TYPE ST_CartUIData :
STRUCT
	m_joystickDataFromUI:ARRAY [0..21] OF USINT;
	m_ctrlEnableFromUI:ST_UI_control;
	m_standColumnHightLimit :LREAL;
	m_surgicalSite : UINT;
	m_surgicalLocation : UINT;
	m_cartDrapingState : UINT;
	m_cartDockingState : UINT;
	m_cartSpecificPosDocking : Vec8d;
	m_cartSpecificPosDraping : Vec8d;
END_STRUCT
END_TYPE

(* stored: Version 1.1.0.1, ProductVersion 3.1.4024.11
   DUT ST_CartUIData: Id {8a7b800d-dda3-4ddf-b29a-44439086ce40} *)
